FUNCTION F_TaskStartDcTimeToExt : T_DCTIME64
VAR_INPUT
END_VAR
VAR
END_VAR

F_TaskStartDcTimeToExt := F_DcToExt(F_GetCurDcTaskTime64());

END_FUNCTION

(* stored: Version 1.1.0.1, ProductVersion 3.1.4022.18
   POU F_TaskStartDcTimeToExt: Id {af9dc5c7-0d13-4791-9001-84456674ac2e}, SpecialFunc None *)
